// TIA Portal V17 export
// export: Created 2024-09-02T12:50:29.8726422Z, ExportSetting WithDefaults, DisplayName Totally Integrated Automation Portal, DisplayVersion V17, DisplayName TIA Portal Openness, DisplayVersion V17, DisplayName TIA Portal Version Control Interface, DisplayVersion V17, DisplayName STEP 7 Professional, DisplayVersion V17, DisplayName STEP 7 Safety, DisplayVersion V17, DisplayName WinCC Professional, DisplayVersion V17
TYPE "e_EKS"
// stored: IsFailsafeCompliant false
   STRUCT
      i_EKS_betriebsbereit : Bool;   // EKS ist Betriebsbereit / EKS jest gotowy do pracy
      i_Datentraeger_anwesend : Bool;   // Datenträger ist anwesend / Data carrier is present
      i_Statusbit_2 : Bool;
      i_Statusbit_3 : Bool;
      i_Status_nur_lesen : Bool;
      i_Auftrag_Fehler : Bool;   // es ist ein Fehler beim Bearbeiten eines Auftrags aufgetreten / An error occurred while processing an order.
      i_Auftrag_fertig : Bool;   // Die Auftragsbearbeitung ist beendet / Order processing is complete
      i_Auftrag_in_Bearbeitung : Bool;   // Die Auftragsbearbeitung läuft / Order processing is running
      i_empfangsdaten_1 : Byte;
      i_Empfangs_Daten : Array[1..116] of Char;   // empfangene Daten vom EKS / Data received from the EKS
      i_Seriennummer : Array[1..8] of Byte;   // Seriennummer 8 Stellen vom EKS / Serial number 8 digits from EKS
      res_127 : Byte;
      res_128 : Byte;
   END_STRUCT;
END_TYPE
